PROGRAM MAIN
VAR
    fbStateMachine : FB_StateMachine;
    smCommands : ST_SM_Commands;
END_VAR

fbStateMachine(
    EnableIn := TRUE,
    cfgAutoRun := TRUE,
    Commands := smCommands
);

_1000_PRG_Homing(sm := fbStateMachine);
_3000_PRG_Running(sm := fbStateMachine);
_2000_PRG_Stopping(sm := fbStateMachine);
_5000_PRG_Aborting(sm := fbStateMachine);
_4000_PRG_Pausing(sm := fbStateMachine);
_6000_PRG_Proceeding(sm := fbStateMachine);

END_PROGRAM

(* stored: Version 1.1.0.1, ProductVersion 3.1.4026.12
   POU MAIN: Id {4f4444b9-0fc9-41d2-8d8b-6376a7d4acc5}, SpecialFunc None *)
